Staubli VAL3: cycle_init.pgx

program cycle_init()
// initialization of the cycle
  local num hours
  local num i
  local num index
  local num l_nSize
begin
  //
  // watch all the instructin has been launched
  //
  // init all the mutex
  cycleStatus:bMutex=false
  // reset
  if saveData:bDebug
    logMsg("[DEBUG] CYCLE: INIT Started")
    ? "CYCLE: INIT Started "
  endIf
  //
  // init all the cyclestatus variable
  //
  call cycleStatus:init()
  //
  // reset the cycle DONE
  //
  call processList:init()
  // check the version status
  call cycle_version()
  if saveData:bDebug
    logMsg("[DEBUG] CYCLE: INIT Terminated")
    ? "CYCLE: INIT Terminated"
  endIf
  // reset all the internal BIT
  bWait=false
  bTimeOut=false
end
